# EPICS autosave request: ADPSL/pslApp/Db/PSL_settings.req
file "ADBase_settings.req", P=$(P), R=$(R)
file "NDFile_settings.req", P=$(P), R=$(R)
$(P)$(R)CameraName
$(P)$(R)TIFFComment
